FUNCTION_BLOCK FB_SimulatedTempSensor EXTENDS FB_ComponentBase IMPLEMENTS I_TempSensor
VAR
	_SimulatedHeatingElement: I_HeatingElement;
	_Temp: LREAL := 20;
END_VAR

//{warning 'Add method implementation '}
METHOD CyclicLogic
VAR
	P_elec			: LREAL;			// Electric power for the heater (W)
	k_hw			: LREAL := 65;		// Heater --> Water coupling (W/deg C)
	h_h				: LREAL := 2;		// Heater --> air loss (W/deg C)
	T_ambient		: LREAL := 20;		// Room temperature (deg C)
	m_h				: LREAL := 0.22;	// Mass of the heater (kg)
	c_h				: LREAL := 500;		// Specific heat of heater (J/kg)
	delta_t 		: LREAL := 0.25;		// Change in time per cycle (s)
	h_w				: LREAL := 18;		// Water --> air loss (W/deg C)
	m_w				: LREAL := 0.75;		// Mass of the water (kg)
	c_w				: LREAL := 4180;	// Specific heat of water (J/kg)
END_VAR
VAR_INST
	T_h : LREAL := 20;
	T_w : LREAL := 20;
END_VAR
IF _SimulatedHeatingElement <> 0 THEN
	// Electrical Input
	P_elec := SEL(_SimulatedHeatingElement.isHeating, 0, 1000);
	// Heater Dynamics
	T_h := T_h + ((P_elec - k_hw * (T_h - T_w) - h_h * (T_h - T_ambient)) / (m_h * c_h)) * delta_t;
	// Water Dynamics
	T_w := T_w + ((k_hw * (T_h -T_w) - h_w * (T_w - T_ambient)) / (m_w * c_w)) *delta_t;
	IF T_w > 100 THEN
		T_w := 100;
	END_IF
	
	_Temp := T_w;
END_IF
END_METHOD

PROPERTY SimulatedHeatingElement : I_HeatingElement
GET
SimulatedHeatingElement := _SimulatedHeatingElement;
END_GET
SET
_SimulatedHeatingElement := SimulatedHeatingElement;
END_SET
END_PROPERTY

{warning 'Add property implementation'}
PROPERTY Temp : LREAL
GET
Temp := _Temp;
END_GET
END_PROPERTY

END_FUNCTION_BLOCK

(* stored: Version 1.1.0.1
   POU FB_SimulatedTempSensor: Id {cd48cc99-3f14-419b-aefa-52a9a041945c}, SpecialFunc None
   Method CyclicLogic: Id {2f8062f2-f056-4eac-850e-993fe1f5becc}
   Property SimulatedHeatingElement: Id {997a7bc8-a06c-4410-8441-22fc4feeb9b8}
   Get Get: Id {aa2f3d88-68a0-4733-b647-0da5ae19cdb5}
   Set Set: Id {0ecfcdb9-d488-44b6-996f-4fd2fd94a3f2}
   Property Temp: Id {1c732188-ab85-47a1-9e7e-9be03453dda7}
   Get Get: Id {575ef6f5-45a6-46e9-bbf9-a85163347da2} *)
